// TIA Portal project "APD Gateway Customer Library Source v00_00_01" (V17)
// 00.00.01 - integrated tag tables

(* hardware
DEVICE "S7-1200 station_1"  S7-1200 Station
   slot 0: "Rack_0"  S7-1200 Rack  Rack  V1.0
   slot 1: "customer"  CPU 1215C AC/DC/Rly  6ES7 215-1BG40-0XB0  V4.0
DEVICE "GSD device_1"  GSD.Device.PN
   slot 0: "Rack"  Rack  V1.0
   slot 1: "profinet_to_adp_gateway"  Profinet_to_ADP_Gateway  6ES7 215-1BG40-0XB0  V4.0
      slot 0: "Message"  Message
      slot 1: "Interface"  Interface
         slot 1: "Port 1"  Port 1
         slot 2: "Port 2"  Port 2
*)

// ===== PLC "customer"  CPU 1215C AC/DC/Rly =====

VAR_GLOBAL   // PLC tag table "Line Formatting"
   "Line_0_Font_Size_&_Weight" AT %QB0 : Byte;
   "Line_0_Scroll_Speed" AT %QB1 : Byte;
   "Line_0_Vertical_Alignment" AT %QB2 : Byte;
   "Line_0_Horizontal_Alignment" AT %QB3 : Byte;
   "Line_0_Hold" AT %QB4 : Byte;
   "Line_1_Font_Size_&_Weight" AT %QB5 : Byte;
   "Line_1_Scroll_Speed" AT %QB6 : Byte;
   "Line_1_Vertical_Alignment" AT %QB7 : Byte;
   "Line_1_Horizontal_Alignment" AT %QB8 : Byte;
   "Line_1_Hold" AT %QB9 : Byte;
   "Line_2_Font_Size_&_Weight" AT %QB10 : Byte;
   "Line_2_Scroll_Speed" AT %QB11 : Byte;
   "Line_2_Vertical_Alignment" AT %QB12 : Byte;
   "Line_2_Horizontal_Alignment" AT %QB13 : Byte;
   "Line_2_Hold" AT %QB14 : Byte;
   "Line_3_Font_Size_&_Weight" AT %QB15 : Byte;
   "Line_3_Scroll_Speed" AT %QB16 : Byte;
   "Line_3_Vertical_Alignment" AT %QB17 : Byte;
   "Line_3_Horizontal_Alignment" AT %QB18 : Byte;
   "Line_3_Hold" AT %QB19 : Byte;
   "Line_4_Font_Size_&_Weight" AT %QB20 : Byte;
   "Line_4_Scroll_Speed" AT %QB21 : Byte;
   "Line_4_Vertical_Alignment" AT %QB22 : Byte;
   "Line_4_Horizontal_Alignment" AT %QB23 : Byte;
   "Line_4_Hold" AT %QB24 : Byte;
END_VAR

VAR_GLOBAL   // PLC tag table "Format Segment 0"
   "Format_Segment_0_Font_Size_&_Weight" AT %QB50 : Byte;
   "Format_Segment_0_Scroll_Speed" AT %QB51 : Byte;
   "Format_Segment_0_Vertical_Alignment" AT %QB52 : Byte;
   "Format_Segment_0_Horizontal_Alignment" AT %QB53 : Byte;
   "Format_Segment_0_Text_Byte_0" AT %QB54 : Byte;
   "Format_Segment_0_Text_Byte_1" AT %QB55 : Byte;
   "Format_Segment_0_Text_Byte_2" AT %QB56 : Byte;
   "Format_Segment_0_Text_Byte_3" AT %QB57 : Byte;
   "Format_Segment_0_Text_Byte_4" AT %QB58 : Byte;
   "Format_Segment_0_Text_Byte_5" AT %QB59 : Byte;
   "Format_Segment_0_Text_Byte_6" AT %QB60 : Byte;
   "Format_Segment_0_Text_Byte_7" AT %QB61 : Byte;
   "Format_Segment_0_Text_Byte_8" AT %QB62 : Byte;
   "Format_Segment_0_Text_Byte_9" AT %QB63 : Byte;
   "Format_Segment_0_Text_Byte_10" AT %QB64 : Byte;
   "Format_Segment_0_Text_Byte_11" AT %QB65 : Byte;
   "Format_Segment_0_Text_Byte_12" AT %QB66 : Byte;
   "Format_Segment_0_Text_Byte_13" AT %QB67 : Byte;
   "Format_Segment_0_Text_Byte_14" AT %QB68 : Byte;
   "Format_Segment_0_Text_Byte_15" AT %QB69 : Byte;
   "Format_Segment_0_Text_Byte_16" AT %QB70 : Byte;
   "Format_Segment_0_Text_Byte_17" AT %QB71 : Byte;
   "Format_Segment_0_Text_Byte_18" AT %QB72 : Byte;
   "Format_Segment_0_Text_Byte_19" AT %QB73 : Byte;
   "Format_Segment_0_Text_Byte_20" AT %QB74 : Byte;
   "Format_Segment_0_Text_Byte_21" AT %QB75 : Byte;
   "Format_Segment_0_Text_Byte_22" AT %QB76 : Byte;
   "Format_Segment_0_Text_Byte_23" AT %QB77 : Byte;
   "Format_Segment_0_Text_Byte_24" AT %QB78 : Byte;
   "Format_Segment_0_Text_Byte_25" AT %QB79 : Byte;
   "Format_Segment_0_Text_Byte_26" AT %QB80 : Byte;
   "Format_Segment_0_Text_Byte_27" AT %QB81 : Byte;
   "Format_Segment_0_Text_Byte_28" AT %QB82 : Byte;
   "Format_Segment_0_Text_Byte_29" AT %QB83 : Byte;
   "Format_Segment_0_Text_Byte_30" AT %QB84 : Byte;
   "Format_Segment_0_Text_Byte_31" AT %QB85 : Byte;
   "Format_Segment_0_Text_Byte_32" AT %QB86 : Byte;
   "Format_Segment_0_Text_Byte_33" AT %QB87 : Byte;
   "Format_Segment_0_Text_Byte_34" AT %QB88 : Byte;
   "Format_Segment_0_Text_Byte_35" AT %QB89 : Byte;
   "Format_Segment_0_Text_Byte_36" AT %QB90 : Byte;
   "Format_Segment_0_Text_Byte_37" AT %QB91 : Byte;
   "Format_Segment_0_Text_Byte_38" AT %QB92 : Byte;
   "Format_Segment_0_Text_Byte_39" AT %QB93 : Byte;
   "Format_Segment_0_Text_Byte_40" AT %QB94 : Byte;
   "Format_Segment_0_Text_Byte_41" AT %QB95 : Byte;
   "Format_Segment_0_Text_Byte_42" AT %QB96 : Byte;
   "Format_Segment_0_Text_Byte_43" AT %QB97 : Byte;
   "Format_Segment_0_Text_Byte_44" AT %QB98 : Byte;
   "Format_Segment_0_Text_Byte_45" AT %QB99 : Byte;
END_VAR

VAR_GLOBAL   // PLC tag table "Format Segment 1"
   "Format_Segment_1_Font_Size_&_Weight" AT %QB100 : Byte;
   "Format_Segment_1_Scroll_Speed" AT %QB101 : Byte;
   "Format_Segment_1_Vertical_Alignment" AT %QB102 : Byte;
   "Format_Segment_1_Horizontal_Alignment" AT %QB103 : Byte;
   "Format_Segment_1_Text_Byte_0" AT %QB104 : Byte;
   "Format_Segment_1_Text_Byte_1" AT %QB105 : Byte;
   "Format_Segment_1_Text_Byte_2" AT %QB106 : Byte;
   "Format_Segment_1_Text_Byte_3" AT %QB107 : Byte;
   "Format_Segment_1_Text_Byte_4" AT %QB108 : Byte;
   "Format_Segment_1_Text_Byte_5" AT %QB109 : Byte;
   "Format_Segment_1_Text_Byte_6" AT %QB110 : Byte;
   "Format_Segment_1_Text_Byte_7" AT %QB111 : Byte;
   "Format_Segment_1_Text_Byte_8" AT %QB112 : Byte;
   "Format_Segment_1_Text_Byte_9" AT %QB113 : Byte;
   "Format_Segment_1_Text_Byte_10" AT %QB114 : Byte;
   "Format_Segment_1_Text_Byte_11" AT %QB115 : Byte;
   "Format_Segment_1_Text_Byte_12" AT %QB116 : Byte;
   "Format_Segment_1_Text_Byte_13" AT %QB117 : Byte;
   "Format_Segment_1_Text_Byte_14" AT %QB118 : Byte;
   "Format_Segment_1_Text_Byte_15" AT %QB119 : Byte;
   "Format_Segment_1_Text_Byte_16" AT %QB120 : Byte;
   "Format_Segment_1_Text_Byte_17" AT %QB121 : Byte;
   "Format_Segment_1_Text_Byte_18" AT %QB122 : Byte;
   "Format_Segment_1_Text_Byte_19" AT %QB123 : Byte;
   "Format_Segment_1_Text_Byte_20" AT %QB124 : Byte;
   "Format_Segment_1_Text_Byte_21" AT %QB125 : Byte;
   "Format_Segment_1_Text_Byte_22" AT %QB126 : Byte;
   "Format_Segment_1_Text_Byte_23" AT %QB127 : Byte;
   "Format_Segment_1_Text_Byte_24" AT %QB128 : Byte;
   "Format_Segment_1_Text_Byte_25" AT %QB129 : Byte;
   "Format_Segment_1_Text_Byte_26" AT %QB130 : Byte;
   "Format_Segment_1_Text_Byte_27" AT %QB131 : Byte;
   "Format_Segment_1_Text_Byte_28" AT %QB132 : Byte;
   "Format_Segment_1_Text_Byte_29" AT %QB133 : Byte;
   "Format_Segment_1_Text_Byte_30" AT %QB134 : Byte;
   "Format_Segment_1_Text_Byte_31" AT %QB135 : Byte;
   "Format_Segment_1_Text_Byte_32" AT %QB136 : Byte;
   "Format_Segment_1_Text_Byte_33" AT %QB137 : Byte;
   "Format_Segment_1_Text_Byte_34" AT %QB138 : Byte;
   "Format_Segment_1_Text_Byte_35" AT %QB139 : Byte;
   "Format_Segment_1_Text_Byte_36" AT %QB140 : Byte;
   "Format_Segment_1_Text_Byte_37" AT %QB141 : Byte;
   "Format_Segment_1_Text_Byte_38" AT %QB142 : Byte;
   "Format_Segment_1_Text_Byte_39" AT %QB143 : Byte;
   "Format_Segment_1_Text_Byte_40" AT %QB144 : Byte;
   "Format_Segment_1_Text_Byte_41" AT %QB145 : Byte;
   "Format_Segment_1_Text_Byte_42" AT %QB146 : Byte;
   "Format_Segment_1_Text_Byte_43" AT %QB147 : Byte;
   "Format_Segment_1_Text_Byte_44" AT %QB148 : Byte;
   "Format_Segment_1_Text_Byte_45" AT %QB149 : Byte;
END_VAR

VAR_GLOBAL   // PLC tag table "Format Segment 2"
   "Format_Segment_2_Font_Size_&_Weight" AT %QB150 : Byte;
   "Format_Segment_2_Scroll_Speed" AT %QB151 : Byte;
   "Format_Segment_2_Vertical_Alignment" AT %QB152 : Byte;
   "Format_Segment_2_Horizontal_Alignment" AT %QB153 : Byte;
   "Format_Segment_2_Text_Byte_0" AT %QB154 : Byte;
   "Format_Segment_2_Text_Byte_1" AT %QB155 : Byte;
   "Format_Segment_2_Text_Byte_2" AT %QB156 : Byte;
   "Format_Segment_2_Text_Byte_3" AT %QB157 : Byte;
   "Format_Segment_2_Text_Byte_4" AT %QB158 : Byte;
   "Format_Segment_2_Text_Byte_5" AT %QB159 : Byte;
   "Format_Segment_2_Text_Byte_6" AT %QB160 : Byte;
   "Format_Segment_2_Text_Byte_7" AT %QB161 : Byte;
   "Format_Segment_2_Text_Byte_8" AT %QB162 : Byte;
   "Format_Segment_2_Text_Byte_9" AT %QB163 : Byte;
   "Format_Segment_2_Text_Byte_10" AT %QB164 : Byte;
   "Format_Segment_2_Text_Byte_11" AT %QB165 : Byte;
   "Format_Segment_2_Text_Byte_12" AT %QB166 : Byte;
   "Format_Segment_2_Text_Byte_13" AT %QB167 : Byte;
   "Format_Segment_2_Text_Byte_14" AT %QB168 : Byte;
   "Format_Segment_2_Text_Byte_15" AT %QB169 : Byte;
   "Format_Segment_2_Text_Byte_16" AT %QB170 : Byte;
   "Format_Segment_2_Text_Byte_17" AT %QB171 : Byte;
   "Format_Segment_2_Text_Byte_18" AT %QB172 : Byte;
   "Format_Segment_2_Text_Byte_19" AT %QB173 : Byte;
   "Format_Segment_2_Text_Byte_20" AT %QB174 : Byte;
   "Format_Segment_2_Text_Byte_21" AT %QB175 : Byte;
   "Format_Segment_2_Text_Byte_22" AT %QB176 : Byte;
   "Format_Segment_2_Text_Byte_23" AT %QB177 : Byte;
   "Format_Segment_2_Text_Byte_24" AT %QB178 : Byte;
   "Format_Segment_2_Text_Byte_25" AT %QB179 : Byte;
   "Format_Segment_2_Text_Byte_26" AT %QB180 : Byte;
   "Format_Segment_2_Text_Byte_27" AT %QB181 : Byte;
   "Format_Segment_2_Text_Byte_28" AT %QB182 : Byte;
   "Format_Segment_2_Text_Byte_29" AT %QB183 : Byte;
   "Format_Segment_2_Text_Byte_30" AT %QB184 : Byte;
   "Format_Segment_2_Text_Byte_31" AT %QB185 : Byte;
   "Format_Segment_2_Text_Byte_32" AT %QB186 : Byte;
   "Format_Segment_2_Text_Byte_33" AT %QB187 : Byte;
   "Format_Segment_2_Text_Byte_34" AT %QB188 : Byte;
   "Format_Segment_2_Text_Byte_35" AT %QB189 : Byte;
   "Format_Segment_2_Text_Byte_36" AT %QB190 : Byte;
   "Format_Segment_2_Text_Byte_37" AT %QB191 : Byte;
   "Format_Segment_2_Text_Byte_38" AT %QB192 : Byte;
   "Format_Segment_2_Text_Byte_39" AT %QB193 : Byte;
   "Format_Segment_2_Text_Byte_40" AT %QB194 : Byte;
   "Format_Segment_2_Text_Byte_41" AT %QB195 : Byte;
   "Format_Segment_2_Text_Byte_42" AT %QB196 : Byte;
   "Format_Segment_2_Text_Byte_43" AT %QB197 : Byte;
   "Format_Segment_2_Text_Byte_44" AT %QB198 : Byte;
   "Format_Segment_2_Text_Byte_45" AT %QB199 : Byte;
END_VAR

VAR_GLOBAL   // PLC tag table "Format Segment 3"
   "Format_Segment_3_Font_Size_&_Weight" AT %QB200 : Byte;
   "Format_Segment_3_Scroll_Speed" AT %QB201 : Byte;
   "Format_Segment_3_Vertical_Alignment" AT %QB202 : Byte;
   "Format_Segment_3_Horizontal_Alignment" AT %QB203 : Byte;
   "Format_Segment_3_Text_Byte_0" AT %QB204 : Byte;
   "Format_Segment_3_Text_Byte_1" AT %QB205 : Byte;
   "Format_Segment_3_Text_Byte_2" AT %QB206 : Byte;
   "Format_Segment_3_Text_Byte_3" AT %QB207 : Byte;
   "Format_Segment_3_Text_Byte_4" AT %QB208 : Byte;
   "Format_Segment_3_Text_Byte_5" AT %QB209 : Byte;
   "Format_Segment_3_Text_Byte_6" AT %QB210 : Byte;
   "Format_Segment_3_Text_Byte_7" AT %QB211 : Byte;
   "Format_Segment_3_Text_Byte_8" AT %QB212 : Byte;
   "Format_Segment_3_Text_Byte_9" AT %QB213 : Byte;
   "Format_Segment_3_Text_Byte_10" AT %QB214 : Byte;
   "Format_Segment_3_Text_Byte_11" AT %QB215 : Byte;
   "Format_Segment_3_Text_Byte_12" AT %QB216 : Byte;
   "Format_Segment_3_Text_Byte_13" AT %QB217 : Byte;
   "Format_Segment_3_Text_Byte_14" AT %QB218 : Byte;
   "Format_Segment_3_Text_Byte_15" AT %QB219 : Byte;
   "Format_Segment_3_Text_Byte_16" AT %QB220 : Byte;
   "Format_Segment_3_Text_Byte_17" AT %QB221 : Byte;
   "Format_Segment_3_Text_Byte_18" AT %QB222 : Byte;
   "Format_Segment_3_Text_Byte_19" AT %QB223 : Byte;
   "Format_Segment_3_Text_Byte_20" AT %QB224 : Byte;
   "Format_Segment_3_Text_Byte_21" AT %QB225 : Byte;
   "Format_Segment_3_Text_Byte_22" AT %QB226 : Byte;
   "Format_Segment_3_Text_Byte_23" AT %QB227 : Byte;
   "Format_Segment_3_Text_Byte_24" AT %QB228 : Byte;
   "Format_Segment_3_Text_Byte_25" AT %QB229 : Byte;
   "Format_Segment_3_Text_Byte_26" AT %QB230 : Byte;
   "Format_Segment_3_Text_Byte_27" AT %QB231 : Byte;
   "Format_Segment_3_Text_Byte_28" AT %QB232 : Byte;
   "Format_Segment_3_Text_Byte_29" AT %QB233 : Byte;
   "Format_Segment_3_Text_Byte_30" AT %QB234 : Byte;
   "Format_Segment_3_Text_Byte_31" AT %QB235 : Byte;
   "Format_Segment_3_Text_Byte_32" AT %QB236 : Byte;
   "Format_Segment_3_Text_Byte_33" AT %QB237 : Byte;
   "Format_Segment_3_Text_Byte_34" AT %QB238 : Byte;
   "Format_Segment_3_Text_Byte_35" AT %QB239 : Byte;
   "Format_Segment_3_Text_Byte_36" AT %QB240 : Byte;
   "Format_Segment_3_Text_Byte_37" AT %QB241 : Byte;
   "Format_Segment_3_Text_Byte_38" AT %QB242 : Byte;
   "Format_Segment_3_Text_Byte_39" AT %QB243 : Byte;
   "Format_Segment_3_Text_Byte_40" AT %QB244 : Byte;
   "Format_Segment_3_Text_Byte_41" AT %QB245 : Byte;
   "Format_Segment_3_Text_Byte_42" AT %QB246 : Byte;
   "Format_Segment_3_Text_Byte_43" AT %QB247 : Byte;
   "Format_Segment_3_Text_Byte_44" AT %QB248 : Byte;
   "Format_Segment_3_Text_Byte_45" AT %QB249 : Byte;
END_VAR

VAR_GLOBAL   // PLC tag table "Format Segment 4"
   "Format_Segment_4_Font_Size_&_Weight" AT %QB250 : Byte;
   "Format_Segment_4_Scroll_Speed" AT %QB251 : Byte;
   "Format_Segment_4_Vertical_Alignment" AT %QB252 : Byte;
   "Format_Segment_4_Horizontal_Alignment" AT %QB253 : Byte;
   "Format_Segment_4_Text_Byte_0" AT %QB254 : Byte;
   "Format_Segment_4_Text_Byte_1" AT %QB255 : Byte;
   "Format_Segment_4_Text_Byte_2" AT %QB256 : Byte;
   "Format_Segment_4_Text_Byte_3" AT %QB257 : Byte;
   "Format_Segment_4_Text_Byte_4" AT %QB258 : Byte;
   "Format_Segment_4_Text_Byte_5" AT %QB259 : Byte;
   "Format_Segment_4_Text_Byte_6" AT %QB260 : Byte;
   "Format_Segment_4_Text_Byte_7" AT %QB261 : Byte;
   "Format_Segment_4_Text_Byte_8" AT %QB262 : Byte;
   "Format_Segment_4_Text_Byte_9" AT %QB263 : Byte;
   "Format_Segment_4_Text_Byte_10" AT %QB264 : Byte;
   "Format_Segment_4_Text_Byte_11" AT %QB265 : Byte;
   "Format_Segment_4_Text_Byte_12" AT %QB266 : Byte;
   "Format_Segment_4_Text_Byte_13" AT %QB267 : Byte;
   "Format_Segment_4_Text_Byte_14" AT %QB268 : Byte;
   "Format_Segment_4_Text_Byte_15" AT %QB269 : Byte;
   "Format_Segment_4_Text_Byte_16" AT %QB270 : Byte;
   "Format_Segment_4_Text_Byte_17" AT %QB271 : Byte;
   "Format_Segment_4_Text_Byte_18" AT %QB272 : Byte;
   "Format_Segment_4_Text_Byte_19" AT %QB273 : Byte;
   "Format_Segment_4_Text_Byte_20" AT %QB274 : Byte;
   "Format_Segment_4_Text_Byte_21" AT %QB275 : Byte;
   "Format_Segment_4_Text_Byte_22" AT %QB276 : Byte;
   "Format_Segment_4_Text_Byte_23" AT %QB277 : Byte;
   "Format_Segment_4_Text_Byte_24" AT %QB278 : Byte;
   "Format_Segment_4_Text_Byte_25" AT %QB279 : Byte;
   "Format_Segment_4_Text_Byte_26" AT %QB280 : Byte;
   "Format_Segment_4_Text_Byte_27" AT %QB281 : Byte;
   "Format_Segment_4_Text_Byte_28" AT %QB282 : Byte;
   "Format_Segment_4_Text_Byte_29" AT %QB283 : Byte;
   "Format_Segment_4_Text_Byte_30" AT %QB284 : Byte;
   "Format_Segment_4_Text_Byte_31" AT %QB285 : Byte;
   "Format_Segment_4_Text_Byte_32" AT %QB286 : Byte;
   "Format_Segment_4_Text_Byte_33" AT %QB287 : Byte;
   "Format_Segment_4_Text_Byte_34" AT %QB288 : Byte;
   "Format_Segment_4_Text_Byte_35" AT %QB289 : Byte;
   "Format_Segment_4_Text_Byte_36" AT %QB290 : Byte;
   "Format_Segment_4_Text_Byte_37" AT %QB291 : Byte;
   "Format_Segment_4_Text_Byte_38" AT %QB292 : Byte;
   "Format_Segment_4_Text_Byte_39" AT %QB293 : Byte;
   "Format_Segment_4_Text_Byte_40" AT %QB294 : Byte;
   "Format_Segment_4_Text_Byte_41" AT %QB295 : Byte;
   "Format_Segment_4_Text_Byte_42" AT %QB296 : Byte;
   "Format_Segment_4_Text_Byte_43" AT %QB297 : Byte;
   "Format_Segment_4_Text_Byte_44" AT %QB298 : Byte;
   "Format_Segment_4_Text_Byte_45" AT %QB299 : Byte;
END_VAR

VAR_GLOBAL   // PLC tag table "Format Segment 5"
   "Format_Segment_5_Font_Size_&_Weight" AT %QB300 : Byte;
   "Format_Segment_5_Scroll_Speed" AT %QB301 : Byte;
   "Format_Segment_5_Vertical_Alignment" AT %QB302 : Byte;
   "Format_Segment_5_Horizontal_Alignment" AT %QB303 : Byte;
   "Format_Segment_5_Text_Byte_0" AT %QB304 : Byte;
   "Format_Segment_5_Text_Byte_1" AT %QB305 : Byte;
   "Format_Segment_5_Text_Byte_2" AT %QB306 : Byte;
   "Format_Segment_5_Text_Byte_3" AT %QB307 : Byte;
   "Format_Segment_5_Text_Byte_4" AT %QB308 : Byte;
   "Format_Segment_5_Text_Byte_5" AT %QB309 : Byte;
   "Format_Segment_5_Text_Byte_6" AT %QB310 : Byte;
   "Format_Segment_5_Text_Byte_7" AT %QB311 : Byte;
   "Format_Segment_5_Text_Byte_8" AT %QB312 : Byte;
   "Format_Segment_5_Text_Byte_9" AT %QB313 : Byte;
   "Format_Segment_5_Text_Byte_10" AT %QB314 : Byte;
   "Format_Segment_5_Text_Byte_11" AT %QB315 : Byte;
   "Format_Segment_5_Text_Byte_12" AT %QB316 : Byte;
   "Format_Segment_5_Text_Byte_13" AT %QB317 : Byte;
   "Format_Segment_5_Text_Byte_14" AT %QB318 : Byte;
   "Format_Segment_5_Text_Byte_15" AT %QB319 : Byte;
   "Format_Segment_5_Text_Byte_16" AT %QB320 : Byte;
   "Format_Segment_5_Text_Byte_17" AT %QB321 : Byte;
   "Format_Segment_5_Text_Byte_18" AT %QB322 : Byte;
   "Format_Segment_5_Text_Byte_19" AT %QB323 : Byte;
   "Format_Segment_5_Text_Byte_20" AT %QB324 : Byte;
   "Format_Segment_5_Text_Byte_21" AT %QB325 : Byte;
   "Format_Segment_5_Text_Byte_22" AT %QB326 : Byte;
   "Format_Segment_5_Text_Byte_23" AT %QB327 : Byte;
   "Format_Segment_5_Text_Byte_24" AT %QB328 : Byte;
   "Format_Segment_5_Text_Byte_25" AT %QB329 : Byte;
   "Format_Segment_5_Text_Byte_26" AT %QB330 : Byte;
   "Format_Segment_5_Text_Byte_27" AT %QB331 : Byte;
   "Format_Segment_5_Text_Byte_28" AT %QB332 : Byte;
   "Format_Segment_5_Text_Byte_29" AT %QB333 : Byte;
   "Format_Segment_5_Text_Byte_30" AT %QB334 : Byte;
   "Format_Segment_5_Text_Byte_31" AT %QB335 : Byte;
   "Format_Segment_5_Text_Byte_32" AT %QB336 : Byte;
   "Format_Segment_5_Text_Byte_33" AT %QB337 : Byte;
   "Format_Segment_5_Text_Byte_34" AT %QB338 : Byte;
   "Format_Segment_5_Text_Byte_35" AT %QB339 : Byte;
   "Format_Segment_5_Text_Byte_36" AT %QB340 : Byte;
   "Format_Segment_5_Text_Byte_37" AT %QB341 : Byte;
   "Format_Segment_5_Text_Byte_38" AT %QB342 : Byte;
   "Format_Segment_5_Text_Byte_39" AT %QB343 : Byte;
   "Format_Segment_5_Text_Byte_40" AT %QB344 : Byte;
   "Format_Segment_5_Text_Byte_41" AT %QB345 : Byte;
   "Format_Segment_5_Text_Byte_42" AT %QB346 : Byte;
   "Format_Segment_5_Text_Byte_43" AT %QB347 : Byte;
   "Format_Segment_5_Text_Byte_44" AT %QB348 : Byte;
   "Format_Segment_5_Text_Byte_45" AT %QB349 : Byte;
END_VAR

VAR_GLOBAL   // PLC tag table "Format Segment 6"
   "Format_Segment_6_Font_Size_&_Weight" AT %QB350 : Byte;
   "Format_Segment_6_Scroll_Speed" AT %QB351 : Byte;
   "Format_Segment_6_Vertical_Alignment" AT %QB352 : Byte;
   "Format_Segment_6_Horizontal_Alignment" AT %QB353 : Byte;
   "Format_Segment_6_Text_Byte_0" AT %QB354 : Byte;
   "Format_Segment_6_Text_Byte_1" AT %QB355 : Byte;
   "Format_Segment_6_Text_Byte_2" AT %QB356 : Byte;
   "Format_Segment_6_Text_Byte_3" AT %QB357 : Byte;
   "Format_Segment_6_Text_Byte_4" AT %QB358 : Byte;
   "Format_Segment_6_Text_Byte_5" AT %QB359 : Byte;
   "Format_Segment_6_Text_Byte_6" AT %QB360 : Byte;
   "Format_Segment_6_Text_Byte_7" AT %QB361 : Byte;
   "Format_Segment_6_Text_Byte_8" AT %QB362 : Byte;
   "Format_Segment_6_Text_Byte_9" AT %QB363 : Byte;
   "Format_Segment_6_Text_Byte_10" AT %QB364 : Byte;
   "Format_Segment_6_Text_Byte_11" AT %QB365 : Byte;
   "Format_Segment_6_Text_Byte_12" AT %QB366 : Byte;
   "Format_Segment_6_Text_Byte_13" AT %QB367 : Byte;
   "Format_Segment_6_Text_Byte_14" AT %QB368 : Byte;
   "Format_Segment_6_Text_Byte_15" AT %QB369 : Byte;
   "Format_Segment_6_Text_Byte_16" AT %QB370 : Byte;
   "Format_Segment_6_Text_Byte_17" AT %QB371 : Byte;
   "Format_Segment_6_Text_Byte_18" AT %QB372 : Byte;
   "Format_Segment_6_Text_Byte_19" AT %QB373 : Byte;
   "Format_Segment_6_Text_Byte_20" AT %QB374 : Byte;
   "Format_Segment_6_Text_Byte_21" AT %QB375 : Byte;
   "Format_Segment_6_Text_Byte_22" AT %QB376 : Byte;
   "Format_Segment_6_Text_Byte_23" AT %QB377 : Byte;
   "Format_Segment_6_Text_Byte_24" AT %QB378 : Byte;
   "Format_Segment_6_Text_Byte_25" AT %QB379 : Byte;
   "Format_Segment_6_Text_Byte_26" AT %QB380 : Byte;
   "Format_Segment_6_Text_Byte_27" AT %QB381 : Byte;
   "Format_Segment_6_Text_Byte_28" AT %QB382 : Byte;
   "Format_Segment_6_Text_Byte_29" AT %QB383 : Byte;
   "Format_Segment_6_Text_Byte_30" AT %QB384 : Byte;
   "Format_Segment_6_Text_Byte_31" AT %QB385 : Byte;
   "Format_Segment_6_Text_Byte_32" AT %QB386 : Byte;
   "Format_Segment_6_Text_Byte_33" AT %QB387 : Byte;
   "Format_Segment_6_Text_Byte_34" AT %QB388 : Byte;
   "Format_Segment_6_Text_Byte_35" AT %QB389 : Byte;
   "Format_Segment_6_Text_Byte_36" AT %QB390 : Byte;
   "Format_Segment_6_Text_Byte_37" AT %QB391 : Byte;
   "Format_Segment_6_Text_Byte_38" AT %QB392 : Byte;
   "Format_Segment_6_Text_Byte_39" AT %QB393 : Byte;
   "Format_Segment_6_Text_Byte_40" AT %QB394 : Byte;
   "Format_Segment_6_Text_Byte_41" AT %QB395 : Byte;
   "Format_Segment_6_Text_Byte_42" AT %QB396 : Byte;
   "Format_Segment_6_Text_Byte_43" AT %QB397 : Byte;
   "Format_Segment_6_Text_Byte_44" AT %QB398 : Byte;
   "Format_Segment_6_Text_Byte_45" AT %QB399 : Byte;
END_VAR

VAR_GLOBAL   // PLC tag table "Format Segment 7"
   "Format_Segment_7_Font_Size_&_Weight" AT %QB400 : Byte;
   "Format_Segment_7_Scroll_Speed" AT %QB401 : Byte;
   "Format_Segment_7_Vertical_Alignment" AT %QB402 : Byte;
   "Format_Segment_7_Horizontal_Alignment" AT %QB403 : Byte;
   "Format_Segment_7_Text_Byte_0" AT %QB404 : Byte;
   "Format_Segment_7_Text_Byte_1" AT %QB405 : Byte;
   "Format_Segment_7_Text_Byte_2" AT %QB406 : Byte;
   "Format_Segment_7_Text_Byte_3" AT %QB407 : Byte;
   "Format_Segment_7_Text_Byte_4" AT %QB408 : Byte;
   "Format_Segment_7_Text_Byte_5" AT %QB409 : Byte;
   "Format_Segment_7_Text_Byte_6" AT %QB410 : Byte;
   "Format_Segment_7_Text_Byte_7" AT %QB411 : Byte;
   "Format_Segment_7_Text_Byte_8" AT %QB412 : Byte;
   "Format_Segment_7_Text_Byte_9" AT %QB413 : Byte;
   "Format_Segment_7_Text_Byte_10" AT %QB414 : Byte;
   "Format_Segment_7_Text_Byte_11" AT %QB415 : Byte;
   "Format_Segment_7_Text_Byte_12" AT %QB416 : Byte;
   "Format_Segment_7_Text_Byte_13" AT %QB417 : Byte;
   "Format_Segment_7_Text_Byte_14" AT %QB418 : Byte;
   "Format_Segment_7_Text_Byte_15" AT %QB419 : Byte;
   "Format_Segment_7_Text_Byte_16" AT %QB420 : Byte;
   "Format_Segment_7_Text_Byte_17" AT %QB421 : Byte;
   "Format_Segment_7_Text_Byte_18" AT %QB422 : Byte;
   "Format_Segment_7_Text_Byte_19" AT %QB423 : Byte;
   "Format_Segment_7_Text_Byte_20" AT %QB424 : Byte;
   "Format_Segment_7_Text_Byte_21" AT %QB425 : Byte;
   "Format_Segment_7_Text_Byte_22" AT %QB426 : Byte;
   "Format_Segment_7_Text_Byte_23" AT %QB427 : Byte;
   "Format_Segment_7_Text_Byte_24" AT %QB428 : Byte;
   "Format_Segment_7_Text_Byte_25" AT %QB429 : Byte;
   "Format_Segment_7_Text_Byte_26" AT %QB430 : Byte;
   "Format_Segment_7_Text_Byte_27" AT %QB431 : Byte;
   "Format_Segment_7_Text_Byte_28" AT %QB432 : Byte;
   "Format_Segment_7_Text_Byte_29" AT %QB433 : Byte;
   "Format_Segment_7_Text_Byte_30" AT %QB434 : Byte;
   "Format_Segment_7_Text_Byte_31" AT %QB435 : Byte;
   "Format_Segment_7_Text_Byte_32" AT %QB436 : Byte;
   "Format_Segment_7_Text_Byte_33" AT %QB437 : Byte;
   "Format_Segment_7_Text_Byte_34" AT %QB438 : Byte;
   "Format_Segment_7_Text_Byte_35" AT %QB439 : Byte;
   "Format_Segment_7_Text_Byte_36" AT %QB440 : Byte;
   "Format_Segment_7_Text_Byte_37" AT %QB441 : Byte;
   "Format_Segment_7_Text_Byte_38" AT %QB442 : Byte;
   "Format_Segment_7_Text_Byte_39" AT %QB443 : Byte;
   "Format_Segment_7_Text_Byte_40" AT %QB444 : Byte;
   "Format_Segment_7_Text_Byte_41" AT %QB445 : Byte;
   "Format_Segment_7_Text_Byte_42" AT %QB446 : Byte;
   "Format_Segment_7_Text_Byte_43" AT %QB447 : Byte;
   "Format_Segment_7_Text_Byte_44" AT %QB448 : Byte;
   "Format_Segment_7_Text_Byte_45" AT %QB449 : Byte;
END_VAR

VAR_GLOBAL   // PLC tag table "Format Segment 8"
   "Format_Segment_8_Font_Size_&_Weight" AT %QB450 : Byte;
   "Format_Segment_8_Scroll_Speed" AT %QB451 : Byte;
   "Format_Segment_8_Vertical_Alignment" AT %QB452 : Byte;
   "Format_Segment_8_Horizontal_Alignment" AT %QB453 : Byte;
   "Format_Segment_8_Text_Byte_0" AT %QB454 : Byte;
   "Format_Segment_8_Text_Byte_1" AT %QB455 : Byte;
   "Format_Segment_8_Text_Byte_2" AT %QB456 : Byte;
   "Format_Segment_8_Text_Byte_3" AT %QB457 : Byte;
   "Format_Segment_8_Text_Byte_4" AT %QB458 : Byte;
   "Format_Segment_8_Text_Byte_5" AT %QB459 : Byte;
   "Format_Segment_8_Text_Byte_6" AT %QB460 : Byte;
   "Format_Segment_8_Text_Byte_7" AT %QB461 : Byte;
   "Format_Segment_8_Text_Byte_8" AT %QB462 : Byte;
   "Format_Segment_8_Text_Byte_9" AT %QB463 : Byte;
   "Format_Segment_8_Text_Byte_10" AT %QB464 : Byte;
   "Format_Segment_8_Text_Byte_11" AT %QB465 : Byte;
   "Format_Segment_8_Text_Byte_12" AT %QB466 : Byte;
   "Format_Segment_8_Text_Byte_13" AT %QB467 : Byte;
   "Format_Segment_8_Text_Byte_14" AT %QB468 : Byte;
   "Format_Segment_8_Text_Byte_15" AT %QB469 : Byte;
   "Format_Segment_8_Text_Byte_16" AT %QB470 : Byte;
   "Format_Segment_8_Text_Byte_17" AT %QB471 : Byte;
   "Format_Segment_8_Text_Byte_18" AT %QB472 : Byte;
   "Format_Segment_8_Text_Byte_19" AT %QB473 : Byte;
   "Format_Segment_8_Text_Byte_20" AT %QB474 : Byte;
   "Format_Segment_8_Text_Byte_21" AT %QB475 : Byte;
   "Format_Segment_8_Text_Byte_22" AT %QB476 : Byte;
   "Format_Segment_8_Text_Byte_23" AT %QB477 : Byte;
   "Format_Segment_8_Text_Byte_24" AT %QB478 : Byte;
   "Format_Segment_8_Text_Byte_25" AT %QB479 : Byte;
   "Format_Segment_8_Text_Byte_26" AT %QB480 : Byte;
   "Format_Segment_8_Text_Byte_27" AT %QB481 : Byte;
   "Format_Segment_8_Text_Byte_28" AT %QB482 : Byte;
   "Format_Segment_8_Text_Byte_29" AT %QB483 : Byte;
   "Format_Segment_8_Text_Byte_30" AT %QB484 : Byte;
   "Format_Segment_8_Text_Byte_31" AT %QB485 : Byte;
   "Format_Segment_8_Text_Byte_32" AT %QB486 : Byte;
   "Format_Segment_8_Text_Byte_33" AT %QB487 : Byte;
   "Format_Segment_8_Text_Byte_34" AT %QB488 : Byte;
   "Format_Segment_8_Text_Byte_35" AT %QB489 : Byte;
   "Format_Segment_8_Text_Byte_36" AT %QB490 : Byte;
   "Format_Segment_8_Text_Byte_37" AT %QB491 : Byte;
   "Format_Segment_8_Text_Byte_38" AT %QB492 : Byte;
   "Format_Segment_8_Text_Byte_39" AT %QB493 : Byte;
   "Format_Segment_8_Text_Byte_40" AT %QB494 : Byte;
   "Format_Segment_8_Text_Byte_41" AT %QB495 : Byte;
   "Format_Segment_8_Text_Byte_42" AT %QB496 : Byte;
   "Format_Segment_8_Text_Byte_43" AT %QB497 : Byte;
   "Format_Segment_8_Text_Byte_44" AT %QB498 : Byte;
   "Format_Segment_8_Text_Byte_45" AT %QB499 : Byte;
END_VAR

VAR_GLOBAL   // PLC tag table "Format Segment 9"
   "Format_Segment_9_Font_Size_&_Weight" AT %QB500 : Byte;
   "Format_Segment_9_Scroll_Speed" AT %QB501 : Byte;
   "Format_Segment_9_Vertical_Alignment" AT %QB502 : Byte;
   "Format_Segment_9_Horizontal_Alignment" AT %QB503 : Byte;
   "Format_Segment_9_Text_Byte_0" AT %QB504 : Byte;
   "Format_Segment_9_Text_Byte_1" AT %QB505 : Byte;
   "Format_Segment_9_Text_Byte_2" AT %QB506 : Byte;
   "Format_Segment_9_Text_Byte_3" AT %QB507 : Byte;
   "Format_Segment_9_Text_Byte_4" AT %QB508 : Byte;
   "Format_Segment_9_Text_Byte_5" AT %QB509 : Byte;
   "Format_Segment_9_Text_Byte_6" AT %QB510 : Byte;
   "Format_Segment_9_Text_Byte_7" AT %QB511 : Byte;
   "Format_Segment_9_Text_Byte_8" AT %QB512 : Byte;
   "Format_Segment_9_Text_Byte_9" AT %QB513 : Byte;
   "Format_Segment_9_Text_Byte_10" AT %QB514 : Byte;
   "Format_Segment_9_Text_Byte_11" AT %QB515 : Byte;
   "Format_Segment_9_Text_Byte_12" AT %QB516 : Byte;
   "Format_Segment_9_Text_Byte_13" AT %QB517 : Byte;
   "Format_Segment_9_Text_Byte_14" AT %QB518 : Byte;
   "Format_Segment_9_Text_Byte_15" AT %QB519 : Byte;
   "Format_Segment_9_Text_Byte_16" AT %QB520 : Byte;
   "Format_Segment_9_Text_Byte_17" AT %QB521 : Byte;
   "Format_Segment_9_Text_Byte_18" AT %QB522 : Byte;
   "Format_Segment_9_Text_Byte_19" AT %QB523 : Byte;
   "Format_Segment_9_Text_Byte_20" AT %QB524 : Byte;
   "Format_Segment_9_Text_Byte_21" AT %QB525 : Byte;
   "Format_Segment_9_Text_Byte_22" AT %QB526 : Byte;
   "Format_Segment_9_Text_Byte_23" AT %QB527 : Byte;
   "Format_Segment_9_Text_Byte_24" AT %QB528 : Byte;
   "Format_Segment_9_Text_Byte_25" AT %QB529 : Byte;
   "Format_Segment_9_Text_Byte_26" AT %QB530 : Byte;
   "Format_Segment_9_Text_Byte_27" AT %QB531 : Byte;
   "Format_Segment_9_Text_Byte_28" AT %QB532 : Byte;
   "Format_Segment_9_Text_Byte_29" AT %QB533 : Byte;
   "Format_Segment_9_Text_Byte_30" AT %QB534 : Byte;
   "Format_Segment_9_Text_Byte_31" AT %QB535 : Byte;
   "Format_Segment_9_Text_Byte_32" AT %QB536 : Byte;
   "Format_Segment_9_Text_Byte_33" AT %QB537 : Byte;
   "Format_Segment_9_Text_Byte_34" AT %QB538 : Byte;
   "Format_Segment_9_Text_Byte_35" AT %QB539 : Byte;
   "Format_Segment_9_Text_Byte_36" AT %QB540 : Byte;
   "Format_Segment_9_Text_Byte_37" AT %QB541 : Byte;
   "Format_Segment_9_Text_Byte_38" AT %QB542 : Byte;
   "Format_Segment_9_Text_Byte_39" AT %QB543 : Byte;
   "Format_Segment_9_Text_Byte_40" AT %QB544 : Byte;
   "Format_Segment_9_Text_Byte_41" AT %QB545 : Byte;
   "Format_Segment_9_Text_Byte_42" AT %QB546 : Byte;
   "Format_Segment_9_Text_Byte_43" AT %QB547 : Byte;
   "Format_Segment_9_Text_Byte_44" AT %QB548 : Byte;
   "Format_Segment_9_Text_Byte_45" AT %QB549 : Byte;
END_VAR

VAR_GLOBAL   // PLC tag table "Format Segment 10"
   "Format_Segment_10_Font_Size_&_Weight" AT %QB550 : Byte;
   "Format_Segment_10_Scroll_Speed" AT %QB551 : Byte;
   "Format_Segment_10_Vertical_Alignment" AT %QB552 : Byte;
   "Format_Segment_10_Horizontal_Alignment" AT %QB553 : Byte;
   "Format_Segment_10_Text_Byte_0" AT %QB554 : Byte;
   "Format_Segment_10_Text_Byte_1" AT %QB555 : Byte;
   "Format_Segment_10_Text_Byte_2" AT %QB556 : Byte;
   "Format_Segment_10_Text_Byte_3" AT %QB557 : Byte;
   "Format_Segment_10_Text_Byte_4" AT %QB558 : Byte;
   "Format_Segment_10_Text_Byte_5" AT %QB559 : Byte;
   "Format_Segment_10_Text_Byte_6" AT %QB560 : Byte;
   "Format_Segment_10_Text_Byte_7" AT %QB561 : Byte;
   "Format_Segment_10_Text_Byte_8" AT %QB562 : Byte;
   "Format_Segment_10_Text_Byte_9" AT %QB563 : Byte;
   "Format_Segment_10_Text_Byte_10" AT %QB564 : Byte;
   "Format_Segment_10_Text_Byte_11" AT %QB565 : Byte;
   "Format_Segment_10_Text_Byte_12" AT %QB566 : Byte;
   "Format_Segment_10_Text_Byte_13" AT %QB567 : Byte;
   "Format_Segment_10_Text_Byte_14" AT %QB568 : Byte;
   "Format_Segment_10_Text_Byte_15" AT %QB569 : Byte;
   "Format_Segment_10_Text_Byte_16" AT %QB570 : Byte;
   "Format_Segment_10_Text_Byte_17" AT %QB571 : Byte;
   "Format_Segment_10_Text_Byte_18" AT %QB572 : Byte;
   "Format_Segment_10_Text_Byte_19" AT %QB573 : Byte;
   "Format_Segment_10_Text_Byte_20" AT %QB574 : Byte;
   "Format_Segment_10_Text_Byte_21" AT %QB575 : Byte;
   "Format_Segment_10_Text_Byte_22" AT %QB576 : Byte;
   "Format_Segment_10_Text_Byte_23" AT %QB577 : Byte;
   "Format_Segment_10_Text_Byte_24" AT %QB578 : Byte;
   "Format_Segment_10_Text_Byte_25" AT %QB579 : Byte;
   "Format_Segment_10_Text_Byte_26" AT %QB580 : Byte;
   "Format_Segment_10_Text_Byte_27" AT %QB581 : Byte;
   "Format_Segment_10_Text_Byte_28" AT %QB582 : Byte;
   "Format_Segment_10_Text_Byte_29" AT %QB583 : Byte;
   "Format_Segment_10_Text_Byte_30" AT %QB584 : Byte;
   "Format_Segment_10_Text_Byte_31" AT %QB585 : Byte;
   "Format_Segment_10_Text_Byte_32" AT %QB586 : Byte;
   "Format_Segment_10_Text_Byte_33" AT %QB587 : Byte;
   "Format_Segment_10_Text_Byte_34" AT %QB588 : Byte;
   "Format_Segment_10_Text_Byte_35" AT %QB589 : Byte;
   "Format_Segment_10_Text_Byte_36" AT %QB590 : Byte;
   "Format_Segment_10_Text_Byte_37" AT %QB591 : Byte;
   "Format_Segment_10_Text_Byte_38" AT %QB592 : Byte;
   "Format_Segment_10_Text_Byte_39" AT %QB593 : Byte;
   "Format_Segment_10_Text_Byte_40" AT %QB594 : Byte;
   "Format_Segment_10_Text_Byte_41" AT %QB595 : Byte;
   "Format_Segment_10_Text_Byte_42" AT %QB596 : Byte;
   "Format_Segment_10_Text_Byte_43" AT %QB597 : Byte;
   "Format_Segment_10_Text_Byte_44" AT %QB598 : Byte;
   "Format_Segment_10_Text_Byte_45" AT %QB599 : Byte;
END_VAR

VAR_GLOBAL   // PLC tag table "Format Segment 11"
   "Format_Segment_11_Font_Size_&_Weight" AT %QB600 : Byte;
   "Format_Segment_11_Scroll_Speed" AT %QB601 : Byte;
   "Format_Segment_11_Vertical_Alignment" AT %QB602 : Byte;
   "Format_Segment_11_Horizontal_Alignment" AT %QB603 : Byte;
   "Format_Segment_11_Text_Byte_0" AT %QB604 : Byte;
   "Format_Segment_11_Text_Byte_1" AT %QB605 : Byte;
   "Format_Segment_11_Text_Byte_2" AT %QB606 : Byte;
   "Format_Segment_11_Text_Byte_3" AT %QB607 : Byte;
   "Format_Segment_11_Text_Byte_4" AT %QB608 : Byte;
   "Format_Segment_11_Text_Byte_5" AT %QB609 : Byte;
   "Format_Segment_11_Text_Byte_6" AT %QB610 : Byte;
   "Format_Segment_11_Text_Byte_7" AT %QB611 : Byte;
   "Format_Segment_11_Text_Byte_8" AT %QB612 : Byte;
   "Format_Segment_11_Text_Byte_9" AT %QB613 : Byte;
   "Format_Segment_11_Text_Byte_10" AT %QB614 : Byte;
   "Format_Segment_11_Text_Byte_11" AT %QB615 : Byte;
   "Format_Segment_11_Text_Byte_12" AT %QB616 : Byte;
   "Format_Segment_11_Text_Byte_13" AT %QB617 : Byte;
   "Format_Segment_11_Text_Byte_14" AT %QB618 : Byte;
   "Format_Segment_11_Text_Byte_15" AT %QB619 : Byte;
   "Format_Segment_11_Text_Byte_16" AT %QB620 : Byte;
   "Format_Segment_11_Text_Byte_17" AT %QB621 : Byte;
   "Format_Segment_11_Text_Byte_18" AT %QB622 : Byte;
   "Format_Segment_11_Text_Byte_19" AT %QB623 : Byte;
   "Format_Segment_11_Text_Byte_20" AT %QB624 : Byte;
   "Format_Segment_11_Text_Byte_21" AT %QB625 : Byte;
   "Format_Segment_11_Text_Byte_22" AT %QB626 : Byte;
   "Format_Segment_11_Text_Byte_23" AT %QB627 : Byte;
   "Format_Segment_11_Text_Byte_24" AT %QB628 : Byte;
   "Format_Segment_11_Text_Byte_25" AT %QB629 : Byte;
   "Format_Segment_11_Text_Byte_26" AT %QB630 : Byte;
   "Format_Segment_11_Text_Byte_27" AT %QB631 : Byte;
   "Format_Segment_11_Text_Byte_28" AT %QB632 : Byte;
   "Format_Segment_11_Text_Byte_29" AT %QB633 : Byte;
   "Format_Segment_11_Text_Byte_30" AT %QB634 : Byte;
   "Format_Segment_11_Text_Byte_31" AT %QB635 : Byte;
   "Format_Segment_11_Text_Byte_32" AT %QB636 : Byte;
   "Format_Segment_11_Text_Byte_33" AT %QB637 : Byte;
   "Format_Segment_11_Text_Byte_34" AT %QB638 : Byte;
   "Format_Segment_11_Text_Byte_35" AT %QB639 : Byte;
   "Format_Segment_11_Text_Byte_36" AT %QB640 : Byte;
   "Format_Segment_11_Text_Byte_37" AT %QB641 : Byte;
   "Format_Segment_11_Text_Byte_38" AT %QB642 : Byte;
   "Format_Segment_11_Text_Byte_39" AT %QB643 : Byte;
   "Format_Segment_11_Text_Byte_40" AT %QB644 : Byte;
   "Format_Segment_11_Text_Byte_41" AT %QB645 : Byte;
   "Format_Segment_11_Text_Byte_42" AT %QB646 : Byte;
   "Format_Segment_11_Text_Byte_43" AT %QB647 : Byte;
   "Format_Segment_11_Text_Byte_44" AT %QB648 : Byte;
   "Format_Segment_11_Text_Byte_45" AT %QB649 : Byte;
END_VAR

VAR_GLOBAL   // PLC tag table "Format Segment 12"
   "Format_Segment_12_Font_Size_&_Weight" AT %QB650 : Byte;
   "Format_Segment_12_Scroll_Speed" AT %QB651 : Byte;
   "Format_Segment_12_Vertical_Alignment" AT %QB652 : Byte;
   "Format_Segment_12_Horizontal_Alignment" AT %QB653 : Byte;
   "Format_Segment_12_Text_Byte_0" AT %QB654 : Byte;
   "Format_Segment_12_Text_Byte_1" AT %QB655 : Byte;
   "Format_Segment_12_Text_Byte_2" AT %QB656 : Byte;
   "Format_Segment_12_Text_Byte_3" AT %QB657 : Byte;
   "Format_Segment_12_Text_Byte_4" AT %QB658 : Byte;
   "Format_Segment_12_Text_Byte_5" AT %QB659 : Byte;
   "Format_Segment_12_Text_Byte_6" AT %QB660 : Byte;
   "Format_Segment_12_Text_Byte_7" AT %QB661 : Byte;
   "Format_Segment_12_Text_Byte_8" AT %QB662 : Byte;
   "Format_Segment_12_Text_Byte_9" AT %QB663 : Byte;
   "Format_Segment_12_Text_Byte_10" AT %QB664 : Byte;
   "Format_Segment_12_Text_Byte_11" AT %QB665 : Byte;
   "Format_Segment_12_Text_Byte_12" AT %QB666 : Byte;
   "Format_Segment_12_Text_Byte_13" AT %QB667 : Byte;
   "Format_Segment_12_Text_Byte_14" AT %QB668 : Byte;
   "Format_Segment_12_Text_Byte_15" AT %QB669 : Byte;
   "Format_Segment_12_Text_Byte_16" AT %QB670 : Byte;
   "Format_Segment_12_Text_Byte_17" AT %QB671 : Byte;
   "Format_Segment_12_Text_Byte_18" AT %QB672 : Byte;
   "Format_Segment_12_Text_Byte_19" AT %QB673 : Byte;
   "Format_Segment_12_Text_Byte_20" AT %QB674 : Byte;
   "Format_Segment_12_Text_Byte_21" AT %QB675 : Byte;
   "Format_Segment_12_Text_Byte_22" AT %QB676 : Byte;
   "Format_Segment_12_Text_Byte_23" AT %QB677 : Byte;
   "Format_Segment_12_Text_Byte_24" AT %QB678 : Byte;
   "Format_Segment_12_Text_Byte_25" AT %QB679 : Byte;
   "Format_Segment_12_Text_Byte_26" AT %QB680 : Byte;
   "Format_Segment_12_Text_Byte_27" AT %QB681 : Byte;
   "Format_Segment_12_Text_Byte_28" AT %QB682 : Byte;
   "Format_Segment_12_Text_Byte_29" AT %QB683 : Byte;
   "Format_Segment_12_Text_Byte_30" AT %QB684 : Byte;
   "Format_Segment_12_Text_Byte_31" AT %QB685 : Byte;
   "Format_Segment_12_Text_Byte_32" AT %QB686 : Byte;
   "Format_Segment_12_Text_Byte_33" AT %QB687 : Byte;
   "Format_Segment_12_Text_Byte_34" AT %QB688 : Byte;
   "Format_Segment_12_Text_Byte_35" AT %QB689 : Byte;
   "Format_Segment_12_Text_Byte_36" AT %QB690 : Byte;
   "Format_Segment_12_Text_Byte_37" AT %QB691 : Byte;
   "Format_Segment_12_Text_Byte_38" AT %QB692 : Byte;
   "Format_Segment_12_Text_Byte_39" AT %QB693 : Byte;
   "Format_Segment_12_Text_Byte_40" AT %QB694 : Byte;
   "Format_Segment_12_Text_Byte_41" AT %QB695 : Byte;
   "Format_Segment_12_Text_Byte_42" AT %QB696 : Byte;
   "Format_Segment_12_Text_Byte_43" AT %QB697 : Byte;
   "Format_Segment_12_Text_Byte_44" AT %QB698 : Byte;
   "Format_Segment_12_Text_Byte_45" AT %QB699 : Byte;
END_VAR

VAR_GLOBAL   // PLC tag table "Format Segment 13"
   "Format_Segment_13_Font_Size_&_Weight" AT %QB700 : Byte;
   "Format_Segment_13_Scroll_Speed" AT %QB701 : Byte;
   "Format_Segment_13_Vertical_Alignment" AT %QB702 : Byte;
   "Format_Segment_13_Horizontal_Alignment" AT %QB703 : Byte;
   "Format_Segment_13_Text_Byte_0" AT %QB704 : Byte;
   "Format_Segment_13_Text_Byte_1" AT %QB705 : Byte;
   "Format_Segment_13_Text_Byte_2" AT %QB706 : Byte;
   "Format_Segment_13_Text_Byte_3" AT %QB707 : Byte;
   "Format_Segment_13_Text_Byte_4" AT %QB708 : Byte;
   "Format_Segment_13_Text_Byte_5" AT %QB709 : Byte;
   "Format_Segment_13_Text_Byte_6" AT %QB710 : Byte;
   "Format_Segment_13_Text_Byte_7" AT %QB711 : Byte;
   "Format_Segment_13_Text_Byte_8" AT %QB712 : Byte;
   "Format_Segment_13_Text_Byte_9" AT %QB713 : Byte;
   "Format_Segment_13_Text_Byte_10" AT %QB714 : Byte;
   "Format_Segment_13_Text_Byte_11" AT %QB715 : Byte;
   "Format_Segment_13_Text_Byte_12" AT %QB716 : Byte;
   "Format_Segment_13_Text_Byte_13" AT %QB717 : Byte;
   "Format_Segment_13_Text_Byte_14" AT %QB718 : Byte;
   "Format_Segment_13_Text_Byte_15" AT %QB719 : Byte;
   "Format_Segment_13_Text_Byte_16" AT %QB720 : Byte;
   "Format_Segment_13_Text_Byte_17" AT %QB721 : Byte;
   "Format_Segment_13_Text_Byte_18" AT %QB722 : Byte;
   "Format_Segment_13_Text_Byte_19" AT %QB723 : Byte;
   "Format_Segment_13_Text_Byte_20" AT %QB724 : Byte;
   "Format_Segment_13_Text_Byte_21" AT %QB725 : Byte;
   "Format_Segment_13_Text_Byte_22" AT %QB726 : Byte;
   "Format_Segment_13_Text_Byte_23" AT %QB727 : Byte;
   "Format_Segment_13_Text_Byte_24" AT %QB728 : Byte;
   "Format_Segment_13_Text_Byte_25" AT %QB729 : Byte;
   "Format_Segment_13_Text_Byte_26" AT %QB730 : Byte;
   "Format_Segment_13_Text_Byte_27" AT %QB731 : Byte;
   "Format_Segment_13_Text_Byte_28" AT %QB732 : Byte;
   "Format_Segment_13_Text_Byte_29" AT %QB733 : Byte;
   "Format_Segment_13_Text_Byte_30" AT %QB734 : Byte;
   "Format_Segment_13_Text_Byte_31" AT %QB735 : Byte;
   "Format_Segment_13_Text_Byte_32" AT %QB736 : Byte;
   "Format_Segment_13_Text_Byte_33" AT %QB737 : Byte;
   "Format_Segment_13_Text_Byte_34" AT %QB738 : Byte;
   "Format_Segment_13_Text_Byte_35" AT %QB739 : Byte;
   "Format_Segment_13_Text_Byte_36" AT %QB740 : Byte;
   "Format_Segment_13_Text_Byte_37" AT %QB741 : Byte;
   "Format_Segment_13_Text_Byte_38" AT %QB742 : Byte;
   "Format_Segment_13_Text_Byte_39" AT %QB743 : Byte;
   "Format_Segment_13_Text_Byte_40" AT %QB744 : Byte;
   "Format_Segment_13_Text_Byte_41" AT %QB745 : Byte;
   "Format_Segment_13_Text_Byte_42" AT %QB746 : Byte;
   "Format_Segment_13_Text_Byte_43" AT %QB747 : Byte;
   "Format_Segment_13_Text_Byte_44" AT %QB748 : Byte;
   "Format_Segment_13_Text_Byte_45" AT %QB749 : Byte;
END_VAR

VAR_GLOBAL   // PLC tag table "Format Segment 14"
   "Format_Segment_14_Font_Size_&_Weight" AT %QB750 : Byte;
   "Format_Segment_14_Scroll_Speed" AT %QB751 : Byte;
   "Format_Segment_14_Vertical_Alignment" AT %QB752 : Byte;
   "Format_Segment_14_Horizontal_Alignment" AT %QB753 : Byte;
   "Format_Segment_14_Text_Byte_0" AT %QB754 : Byte;
   "Format_Segment_14_Text_Byte_1" AT %QB755 : Byte;
   "Format_Segment_14_Text_Byte_2" AT %QB756 : Byte;
   "Format_Segment_14_Text_Byte_3" AT %QB757 : Byte;
   "Format_Segment_14_Text_Byte_4" AT %QB758 : Byte;
   "Format_Segment_14_Text_Byte_5" AT %QB759 : Byte;
   "Format_Segment_14_Text_Byte_6" AT %QB760 : Byte;
   "Format_Segment_14_Text_Byte_7" AT %QB761 : Byte;
   "Format_Segment_14_Text_Byte_8" AT %QB762 : Byte;
   "Format_Segment_14_Text_Byte_9" AT %QB763 : Byte;
   "Format_Segment_14_Text_Byte_10" AT %QB764 : Byte;
   "Format_Segment_14_Text_Byte_11" AT %QB765 : Byte;
   "Format_Segment_14_Text_Byte_12" AT %QB766 : Byte;
   "Format_Segment_14_Text_Byte_13" AT %QB767 : Byte;
   "Format_Segment_14_Text_Byte_14" AT %QB768 : Byte;
   "Format_Segment_14_Text_Byte_15" AT %QB769 : Byte;
   "Format_Segment_14_Text_Byte_16" AT %QB770 : Byte;
   "Format_Segment_14_Text_Byte_17" AT %QB771 : Byte;
   "Format_Segment_14_Text_Byte_18" AT %QB772 : Byte;
   "Format_Segment_14_Text_Byte_19" AT %QB773 : Byte;
   "Format_Segment_14_Text_Byte_20" AT %QB774 : Byte;
   "Format_Segment_14_Text_Byte_21" AT %QB775 : Byte;
   "Format_Segment_14_Text_Byte_22" AT %QB776 : Byte;
   "Format_Segment_14_Text_Byte_23" AT %QB777 : Byte;
   "Format_Segment_14_Text_Byte_24" AT %QB778 : Byte;
   "Format_Segment_14_Text_Byte_25" AT %QB779 : Byte;
   "Format_Segment_14_Text_Byte_26" AT %QB780 : Byte;
   "Format_Segment_14_Text_Byte_27" AT %QB781 : Byte;
   "Format_Segment_14_Text_Byte_28" AT %QB782 : Byte;
   "Format_Segment_14_Text_Byte_29" AT %QB783 : Byte;
   "Format_Segment_14_Text_Byte_30" AT %QB784 : Byte;
   "Format_Segment_14_Text_Byte_31" AT %QB785 : Byte;
   "Format_Segment_14_Text_Byte_32" AT %QB786 : Byte;
   "Format_Segment_14_Text_Byte_33" AT %QB787 : Byte;
   "Format_Segment_14_Text_Byte_34" AT %QB788 : Byte;
   "Format_Segment_14_Text_Byte_35" AT %QB789 : Byte;
   "Format_Segment_14_Text_Byte_36" AT %QB790 : Byte;
   "Format_Segment_14_Text_Byte_37" AT %QB791 : Byte;
   "Format_Segment_14_Text_Byte_38" AT %QB792 : Byte;
   "Format_Segment_14_Text_Byte_39" AT %QB793 : Byte;
   "Format_Segment_14_Text_Byte_40" AT %QB794 : Byte;
   "Format_Segment_14_Text_Byte_41" AT %QB795 : Byte;
   "Format_Segment_14_Text_Byte_42" AT %QB796 : Byte;
   "Format_Segment_14_Text_Byte_43" AT %QB797 : Byte;
   "Format_Segment_14_Text_Byte_44" AT %QB798 : Byte;
   "Format_Segment_14_Text_Byte_45" AT %QB799 : Byte;
END_VAR

VAR_GLOBAL   // PLC tag table "Format Segment 15"
   "Format_Segment_15_Font_Size_&_Weight" AT %QB800 : Byte;
   "Format_Segment_15_Scroll_Speed" AT %QB801 : Byte;
   "Format_Segment_15_Vertical_Alignment" AT %QB802 : Byte;
   "Format_Segment_15_Horizontal_Alignment" AT %QB803 : Byte;
   "Format_Segment_15_Text_Byte_0" AT %QB804 : Byte;
   "Format_Segment_15_Text_Byte_1" AT %QB805 : Byte;
   "Format_Segment_15_Text_Byte_2" AT %QB806 : Byte;
   "Format_Segment_15_Text_Byte_3" AT %QB807 : Byte;
   "Format_Segment_15_Text_Byte_4" AT %QB808 : Byte;
   "Format_Segment_15_Text_Byte_5" AT %QB809 : Byte;
   "Format_Segment_15_Text_Byte_6" AT %QB810 : Byte;
   "Format_Segment_15_Text_Byte_7" AT %QB811 : Byte;
   "Format_Segment_15_Text_Byte_8" AT %QB812 : Byte;
   "Format_Segment_15_Text_Byte_9" AT %QB813 : Byte;
   "Format_Segment_15_Text_Byte_10" AT %QB814 : Byte;
   "Format_Segment_15_Text_Byte_11" AT %QB815 : Byte;
   "Format_Segment_15_Text_Byte_12" AT %QB816 : Byte;
   "Format_Segment_15_Text_Byte_13" AT %QB817 : Byte;
   "Format_Segment_15_Text_Byte_14" AT %QB818 : Byte;
   "Format_Segment_15_Text_Byte_15" AT %QB819 : Byte;
   "Format_Segment_15_Text_Byte_16" AT %QB820 : Byte;
   "Format_Segment_15_Text_Byte_17" AT %QB821 : Byte;
   "Format_Segment_15_Text_Byte_18" AT %QB822 : Byte;
   "Format_Segment_15_Text_Byte_19" AT %QB823 : Byte;
   "Format_Segment_15_Text_Byte_20" AT %QB824 : Byte;
   "Format_Segment_15_Text_Byte_21" AT %QB825 : Byte;
   "Format_Segment_15_Text_Byte_22" AT %QB826 : Byte;
   "Format_Segment_15_Text_Byte_23" AT %QB827 : Byte;
   "Format_Segment_15_Text_Byte_24" AT %QB828 : Byte;
   "Format_Segment_15_Text_Byte_25" AT %QB829 : Byte;
   "Format_Segment_15_Text_Byte_26" AT %QB830 : Byte;
   "Format_Segment_15_Text_Byte_27" AT %QB831 : Byte;
   "Format_Segment_15_Text_Byte_28" AT %QB832 : Byte;
   "Format_Segment_15_Text_Byte_29" AT %QB833 : Byte;
   "Format_Segment_15_Text_Byte_30" AT %QB834 : Byte;
   "Format_Segment_15_Text_Byte_31" AT %QB835 : Byte;
   "Format_Segment_15_Text_Byte_32" AT %QB836 : Byte;
   "Format_Segment_15_Text_Byte_33" AT %QB837 : Byte;
   "Format_Segment_15_Text_Byte_34" AT %QB838 : Byte;
   "Format_Segment_15_Text_Byte_35" AT %QB839 : Byte;
   "Format_Segment_15_Text_Byte_36" AT %QB840 : Byte;
   "Format_Segment_15_Text_Byte_37" AT %QB841 : Byte;
   "Format_Segment_15_Text_Byte_38" AT %QB842 : Byte;
   "Format_Segment_15_Text_Byte_39" AT %QB843 : Byte;
   "Format_Segment_15_Text_Byte_40" AT %QB844 : Byte;
   "Format_Segment_15_Text_Byte_41" AT %QB845 : Byte;
   "Format_Segment_15_Text_Byte_42" AT %QB846 : Byte;
   "Format_Segment_15_Text_Byte_43" AT %QB847 : Byte;
   "Format_Segment_15_Text_Byte_44" AT %QB848 : Byte;
   "Format_Segment_15_Text_Byte_45" AT %QB849 : Byte;
END_VAR

VAR_GLOBAL   // PLC tag table "Format Segment 16"
   "Format_Segment_16_Font_Size_&_Weight" AT %QB850 : Byte;
   "Format_Segment_16_Scroll_Speed" AT %QB851 : Byte;
   "Format_Segment_16_Vertical_Alignment" AT %QB852 : Byte;
   "Format_Segment_16_Horizontal_Alignment" AT %QB853 : Byte;
   "Format_Segment_16_Text_Byte_0" AT %QB854 : Byte;
   "Format_Segment_16_Text_Byte_1" AT %QB855 : Byte;
   "Format_Segment_16_Text_Byte_2" AT %QB856 : Byte;
   "Format_Segment_16_Text_Byte_3" AT %QB857 : Byte;
   "Format_Segment_16_Text_Byte_4" AT %QB858 : Byte;
   "Format_Segment_16_Text_Byte_5" AT %QB859 : Byte;
   "Format_Segment_16_Text_Byte_6" AT %QB860 : Byte;
   "Format_Segment_16_Text_Byte_7" AT %QB861 : Byte;
   "Format_Segment_16_Text_Byte_8" AT %QB862 : Byte;
   "Format_Segment_16_Text_Byte_9" AT %QB863 : Byte;
   "Format_Segment_16_Text_Byte_10" AT %QB864 : Byte;
   "Format_Segment_16_Text_Byte_11" AT %QB865 : Byte;
   "Format_Segment_16_Text_Byte_12" AT %QB866 : Byte;
   "Format_Segment_16_Text_Byte_13" AT %QB867 : Byte;
   "Format_Segment_16_Text_Byte_14" AT %QB868 : Byte;
   "Format_Segment_16_Text_Byte_15" AT %QB869 : Byte;
   "Format_Segment_16_Text_Byte_16" AT %QB870 : Byte;
   "Format_Segment_16_Text_Byte_17" AT %QB871 : Byte;
   "Format_Segment_16_Text_Byte_18" AT %QB872 : Byte;
   "Format_Segment_16_Text_Byte_19" AT %QB873 : Byte;
   "Format_Segment_16_Text_Byte_20" AT %QB874 : Byte;
   "Format_Segment_16_Text_Byte_21" AT %QB875 : Byte;
   "Format_Segment_16_Text_Byte_22" AT %QB876 : Byte;
   "Format_Segment_16_Text_Byte_23" AT %QB877 : Byte;
   "Format_Segment_16_Text_Byte_24" AT %QB878 : Byte;
   "Format_Segment_16_Text_Byte_25" AT %QB879 : Byte;
   "Format_Segment_16_Text_Byte_26" AT %QB880 : Byte;
   "Format_Segment_16_Text_Byte_27" AT %QB881 : Byte;
   "Format_Segment_16_Text_Byte_28" AT %QB882 : Byte;
   "Format_Segment_16_Text_Byte_29" AT %QB883 : Byte;
   "Format_Segment_16_Text_Byte_30" AT %QB884 : Byte;
   "Format_Segment_16_Text_Byte_31" AT %QB885 : Byte;
   "Format_Segment_16_Text_Byte_32" AT %QB886 : Byte;
   "Format_Segment_16_Text_Byte_33" AT %QB887 : Byte;
   "Format_Segment_16_Text_Byte_34" AT %QB888 : Byte;
   "Format_Segment_16_Text_Byte_35" AT %QB889 : Byte;
   "Format_Segment_16_Text_Byte_36" AT %QB890 : Byte;
   "Format_Segment_16_Text_Byte_37" AT %QB891 : Byte;
   "Format_Segment_16_Text_Byte_38" AT %QB892 : Byte;
   "Format_Segment_16_Text_Byte_39" AT %QB893 : Byte;
   "Format_Segment_16_Text_Byte_40" AT %QB894 : Byte;
   "Format_Segment_16_Text_Byte_41" AT %QB895 : Byte;
   "Format_Segment_16_Text_Byte_42" AT %QB896 : Byte;
   "Format_Segment_16_Text_Byte_43" AT %QB897 : Byte;
   "Format_Segment_16_Text_Byte_44" AT %QB898 : Byte;
   "Format_Segment_16_Text_Byte_45" AT %QB899 : Byte;
END_VAR

VAR_GLOBAL   // PLC tag table "Format Segment 17"
   "Format_Segment_17_Font_Size_&_Weight" AT %QB900 : Byte;
   "Format_Segment_17_Scroll_Speed" AT %QB901 : Byte;
   "Format_Segment_17_Vertical_Alignment" AT %QB902 : Byte;
   "Format_Segment_17_Horizontal_Alignment" AT %QB903 : Byte;
   "Format_Segment_17_Text_Byte_0" AT %QB904 : Byte;
   "Format_Segment_17_Text_Byte_1" AT %QB905 : Byte;
   "Format_Segment_17_Text_Byte_2" AT %QB906 : Byte;
   "Format_Segment_17_Text_Byte_3" AT %QB907 : Byte;
   "Format_Segment_17_Text_Byte_4" AT %QB908 : Byte;
   "Format_Segment_17_Text_Byte_5" AT %QB909 : Byte;
   "Format_Segment_17_Text_Byte_6" AT %QB910 : Byte;
   "Format_Segment_17_Text_Byte_7" AT %QB911 : Byte;
   "Format_Segment_17_Text_Byte_8" AT %QB912 : Byte;
   "Format_Segment_17_Text_Byte_9" AT %QB913 : Byte;
   "Format_Segment_17_Text_Byte_10" AT %QB914 : Byte;
   "Format_Segment_17_Text_Byte_11" AT %QB915 : Byte;
   "Format_Segment_17_Text_Byte_12" AT %QB916 : Byte;
   "Format_Segment_17_Text_Byte_13" AT %QB917 : Byte;
   "Format_Segment_17_Text_Byte_14" AT %QB918 : Byte;
   "Format_Segment_17_Text_Byte_15" AT %QB919 : Byte;
   "Format_Segment_17_Text_Byte_16" AT %QB920 : Byte;
   "Format_Segment_17_Text_Byte_17" AT %QB921 : Byte;
   "Format_Segment_17_Text_Byte_18" AT %QB922 : Byte;
   "Format_Segment_17_Text_Byte_19" AT %QB923 : Byte;
   "Format_Segment_17_Text_Byte_20" AT %QB924 : Byte;
   "Format_Segment_17_Text_Byte_21" AT %QB925 : Byte;
   "Format_Segment_17_Text_Byte_22" AT %QB926 : Byte;
   "Format_Segment_17_Text_Byte_23" AT %QB927 : Byte;
   "Format_Segment_17_Text_Byte_24" AT %QB928 : Byte;
   "Format_Segment_17_Text_Byte_25" AT %QB929 : Byte;
   "Format_Segment_17_Text_Byte_26" AT %QB930 : Byte;
   "Format_Segment_17_Text_Byte_27" AT %QB931 : Byte;
   "Format_Segment_17_Text_Byte_28" AT %QB932 : Byte;
   "Format_Segment_17_Text_Byte_29" AT %QB933 : Byte;
   "Format_Segment_17_Text_Byte_30" AT %QB934 : Byte;
   "Format_Segment_17_Text_Byte_31" AT %QB935 : Byte;
   "Format_Segment_17_Text_Byte_32" AT %QB936 : Byte;
   "Format_Segment_17_Text_Byte_33" AT %QB937 : Byte;
   "Format_Segment_17_Text_Byte_34" AT %QB938 : Byte;
   "Format_Segment_17_Text_Byte_35" AT %QB939 : Byte;
   "Format_Segment_17_Text_Byte_36" AT %QB940 : Byte;
   "Format_Segment_17_Text_Byte_37" AT %QB941 : Byte;
   "Format_Segment_17_Text_Byte_38" AT %QB942 : Byte;
   "Format_Segment_17_Text_Byte_39" AT %QB943 : Byte;
   "Format_Segment_17_Text_Byte_40" AT %QB944 : Byte;
   "Format_Segment_17_Text_Byte_41" AT %QB945 : Byte;
   "Format_Segment_17_Text_Byte_42" AT %QB946 : Byte;
   "Format_Segment_17_Text_Byte_43" AT %QB947 : Byte;
   "Format_Segment_17_Text_Byte_44" AT %QB948 : Byte;
   "Format_Segment_17_Text_Byte_45" AT %QB949 : Byte;
END_VAR

VAR_GLOBAL CONSTANT   // PLC tag table "Constants"
   "FONT_NORMAL_5" : SInt := 1;
   "FONT_NORMAL_7" : SInt := 2;
   "FONT_NORMAL_9" : SInt := 3;
   "FONT_NORMAL_11" : SInt := 4;
   "FONT_NORMAL_14" : SInt := 5;
   "FONT_NORMAL_15" : SInt := 6;
   "FONT_NORMAL_16" : SInt := 7;
   "FONT_NORMAL_22" : SInt := 8;
   "FONT_NORMAL_24" : SInt := 9;
   "FONT_NORMAL_30" : SInt := 10;
   "FONT_NORMAL_32" : SInt := 11;
   "FONT_NORMAL_40" : SInt := 12;
   "FONT_BOLD_5" : SInt := 13;
   "FONT_BOLD_7" : SInt := 14;
   "FONT_BOLD_9" : SInt := 15;
   "FONT_BOLD_11" : SInt := 16;
   "FONT_BOLD_14" : SInt := 17;
   "FONT_BOLD_15" : SInt := 18;
   "FONT_BOLD_16" : SInt := 19;
   "FONT_BOLD_22" : SInt := 20;
   "FONT_BOLD_24" : SInt := 21;
   "FONT_BOLD_30" : SInt := 22;
   "FONT_BOLD_32" : SInt := 23;
   "FONT_BOLD_40" : SInt := 24;
   "SCROLL_FASTEST" : SInt := 1;
   "SCROLL_FAST" : SInt := 2;
   "SCROLL_NORMAL" : SInt := 3;
   "SCROLL_SLOW" : SInt := 4;
   "SCROLL_SLOWEST" : SInt := 5;
   "HORIZONTAL_LEFT" : SInt := 1;
   "HORIZONTAL_RIGHT" : SInt := 2;
   "HORIZONTAL_CENTER" : SInt := 3;
   "VERTICAL_BOTTOM" : SInt := 1;
   "VERTICAL_MIDDLE" : SInt := 2;
   "VERTICAL_TOP" : SInt := 3;
   "VERTICAL_FILL" : SInt := 4;
   "FOREGROUND_COLOR_BLACK" : SInt := 1;
   "FOREGROUND_COLOR_RED" : SInt := 2;
   "FOREGROUND_COLOR_GREEN" : SInt := 3;
   "FOREGROUND_COLOR_YELLOW" : SInt := 4;
   "FOREGROUND_COLOR_MIX_1" : SInt := 5;
   "FOREGROUND_COLOR_MIX_2" : SInt := 6;
   "FOREGROUND_COLOR_MIX_3" : SInt := 7;
   "FOREGROUND_COLOR_MIX_4" : SInt := 8;
   "FOREGROUND_COLOR_BLUE" : SInt := 9;
   "FOREGROUND_COLOR_WHITE" : SInt := 10;
   "BACKGROUND_COLOR_BLACK" : SInt := 1;
   "BACKGROUND_COLOR_RED" : SInt := 2;
   "BACKGROUND_COLOR_GREEN" : SInt := 3;
   "BACKGROUND_COLOR_YELLOW" : SInt := 4;
   "FLASH_ON" : SInt := 1;
   "FLASH_OFF" : SInt := 2;
END_VAR

// folder: ADP Gateway Interface

TYPE "ADP_Gateway_Interface.UDT"
   STRUCT
      hardware_address : DInt;
      line_formats : Array[0..4] of "ADP_Gateway_Interface.Line_Format.UDT";
      format_segments : Array[0..17] of "ADP_Gateway_Interface.Format_Segment.UDT";
   END_STRUCT;
END_TYPE

TYPE "ADP_Gateway_Interface.Line_Format.UDT"
   STRUCT
      font : SInt := 1;
      scroll_speed : SInt := 1;
      vertical_alignment : SInt := 1;
      horizontal_alignment : SInt := 1;
      hold : SInt := 5;
   END_STRUCT;
END_TYPE

TYPE "ADP_Gateway_Interface.Format_Segment.UDT"
   STRUCT
      foreground_color : SInt := 1;
      background_color : SInt := 1;
      flash : SInt := 1;
      line_number : SInt := -1;
      text : String[46];
   END_STRUCT;
END_TYPE

DATA_BLOCK "ADP_Gateway_Interface_Data"   // DB1
{ S7_Optimized_Access := 'TRUE' }
VERSION : 0.1
BEGIN
END_DATA_BLOCK

// folder: (top level)

ORGANIZATION_BLOCK "Main"   // OB1, LAD, ProgramCycle
TITLE = "Main Program Sweep (Cycle)"
{ S7_Optimized_Access := 'TRUE' }
VERSION : 0.1
   VAR_INPUT
      Initial_Call : Bool;   // Initial call of this OB
      Remanence : Bool;   // =True, if remanent data are available
   END_VAR
BEGIN

REGION Network 1 (SCL)
   "ADP_Gateway_Interface_Data".hardware_address := 0;

   "ADP_Gateway_Interface_Data".line_formats[0].font := "FONT_BOLD_14";
   "ADP_Gateway_Interface_Data".line_formats[0].horizontal_alignment := "HORIZONTAL_LEFT";
   "ADP_Gateway_Interface_Data".line_formats[0].scroll_speed := "SCROLL_NORMAL";

   "ADP_Gateway_Interface_Data".format_segments[0].foreground_color := "FOREGROUND_COLOR_RED";
   "ADP_Gateway_Interface_Data".format_segments[0].flash := "FLASH_OFF";
END_REGION

REGION Network 2
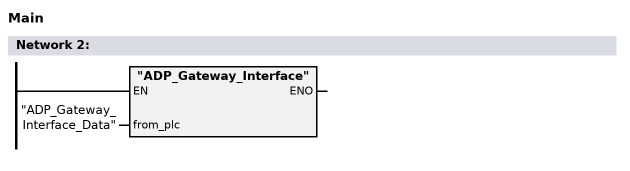
   RUNG wire#powerrail
      "ADP_Gateway_Interface"(from_plc := "ADP_Gateway_Interface_Data")
   END_RUNG
   // the same network as SCL:
   "ADP_Gateway_Interface"(from_plc := "ADP_Gateway_Interface_Data");
END_REGION
END_ORGANIZATION_BLOCK

// folder: ADP Gateway Interface

FUNCTION "ADP_Gateway_Interface" : Void   // FC1, SCL
TITLE = ADP Gateway Interface
{ S7_Optimized_Access := 'TRUE' }
AUTHOR : Machado
VERSION : 0.1
// for use with GSD file version xxxxx
   VAR_INPUT
      from_plc : "ADP_Gateway_Interface.UDT";
   END_VAR
   VAR_TEMP
      i : Int;
   END_VAR
   VAR CONSTANT
      LINE_COUNT : DInt := 4;   // 5 lines, 0 indexed
      FORMAT_SEGMENT_COUNT : DInt := 17;   // 18 format segments, 0 indexed
   END_VAR
BEGIN
   REGION LINE FORMATS
       FOR #i := 0 TO #LINE_COUNT DO
           "ADP_Gateway_Interface.Poke_Line_Formatting"(base_offset := 0,
                                                        from_plc := #from_plc.line_formats[#i],
                                                        line_number := #i);
       END_FOR;
   END_REGION


   REGION FORMAT SEGMENTS
       FOR #i := 0 TO #FORMAT_SEGMENT_COUNT DO
           "ADP_Gateway_Interface.Poke_Format_Segment"(base_offset := 50,
                                                       segment_number := #i,
                                                       format_segment := #from_plc.format_segments[#i]);
       END_FOR;
   END_REGION


   RETURN;
END_FUNCTION

FUNCTION "ADP_Gateway_Interface.Poke_Line_Formatting" : Void   // FC2, SCL
{ S7_Optimized_Access := 'TRUE' }
VERSION : 0.1
   VAR_INPUT
      base_offset : DInt;
      from_plc : "ADP_Gateway_Interface.Line_Format.UDT";
      line_number : Int;
   END_VAR
   VAR_TEMP
      offset : DInt;
   END_VAR
   VAR CONSTANT
      BYTES_PER_LINE : DInt := 5;
      OUTPUT_AREA : Byte := 16#82;
      NO_DB : DInt;
   END_VAR
BEGIN
   REGION BASE OFFSET
       #offset := #line_number * #BYTES_PER_LINE + #base_offset;
   END_REGION


   REGION FONT
       POKE(area := #OUTPUT_AREA,
            dbNumber := #NO_DB,
            byteOffset := #offset,
            value := SINT_TO_BYTE(#from_plc.font));
   END_REGION


   REGION SCROLL SPEED
       POKE(area := #OUTPUT_AREA,
            dbNumber := #NO_DB,
            byteOffset := #offset + 1,
            value := SINT_TO_BYTE(#from_plc.scroll_speed));
   END_REGION


   REGION VERTICAL ALIGNMENT
       POKE(area := #OUTPUT_AREA,
            dbNumber := #NO_DB,
            byteOffset := #offset + 2,
            value := SINT_TO_BYTE(#from_plc.vertical_alignment));
   END_REGION


   REGION HORIZONTAL ALIGNMENT
       POKE(area := #OUTPUT_AREA,
            dbNumber := #NO_DB,
            byteOffset := #offset + 3,
            value := SINT_TO_BYTE(#from_plc.horizontal_alignment));
   END_REGION


   REGION HOLD
       POKE(area := #OUTPUT_AREA,
            dbNumber := #NO_DB,
            byteOffset := #offset + 4,
            value := SINT_TO_BYTE(#from_plc.hold));
   END_REGION


   RETURN;
END_FUNCTION

FUNCTION "ADP_Gateway_Interface.Poke_Format_Segment" : Void   // FC3, SCL
{ S7_Optimized_Access := 'TRUE' }
VERSION : 0.1
   VAR_INPUT
      base_offset : DInt;
      segment_number : DInt;
      format_segment : "ADP_Gateway_Interface.Format_Segment.UDT";
   END_VAR
   VAR_TEMP
      i : DInt;
      offset : DInt;
   END_VAR
   VAR CONSTANT
      BYTES_PER_AREA : DInt := 50;
      BYTES_OF_TEXT : DInt := 49;
      OUTPUT_AREA : Byte := 16#82;
      NO_DB : DInt;
   END_VAR
BEGIN
   REGION BASE OFFSET
       #offset := #base_offset + #segment_number * #BYTES_PER_AREA;
   END_REGION


   REGION FOREGROUND
       POKE(area := #OUTPUT_AREA,
            dbNumber := #NO_DB,
            byteOffset := #offset,
            value := SINT_TO_BYTE(#format_segment.foreground_color));
   END_REGION


   REGION BACKGROUND
       POKE(area := #OUTPUT_AREA,
            dbNumber := #NO_DB,
            byteOffset := #offset + 1,
            value := SINT_TO_BYTE(#format_segment.background_color));
   END_REGION


   REGION FLASH
       POKE(area := #OUTPUT_AREA,
            dbNumber := #NO_DB,
            byteOffset := #offset + 2,
            value := SINT_TO_BYTE(#format_segment.flash));
   END_REGION


   REGION LINE NUMBER
       POKE(area := #OUTPUT_AREA,
            dbNumber := #NO_DB,
            byteOffset := #offset + 3,
            value := SINT_TO_BYTE(#format_segment.line_number));
   END_REGION


   REGION TEXT
       FOR #i := 0 TO #BYTES_OF_TEXT DO
           POKE(area := #OUTPUT_AREA,
                dbNumber := #NO_DB,
                byteOffset := #offset + #i + 4,
                value := CHAR_TO_BYTE(#format_segment.text[#i]));
       END_FOR;
   END_REGION
END_FUNCTION